TYPE (* A Structure with 4 Bits *)
  (* Version 1.0, 2024-02-21, franz *)
  st4b : STRUCT
    b0 : BOOL; (* BIT 00 *)
    b1 : BOOL; (* BIT 01 *)
    b2 : BOOL; (* BIT 02 *)
    b3 : BOOL; (* BIT 03 *)
  END_STRUCT;
END_TYPE
